{attribute 'linkalways'} 
{attribute 'no_explicit_call' := 'This FB is a CLASS and must be accessed using methods or properties'}
{attribute 'enable_dynamic_creation'}
FUNCTION_BLOCK FINAL Node_NOT EXTENDS Node
VAR
	in : _BOOL(FALSE);
	out : _BOOL(FALSE);
END_VAR

METHOD PUBLIC  Clone : I_Node
VAR
	pNode : POINTER TO Node_NOT;
END_VAR
pNode := __NEW(Node_NOT);
Clone := pNode^;
END_METHOD

METHOD FB_init : BOOL
VAR_INPUT
	bInitRetains : BOOL; // if TRUE, the retain variables are initialized (warm start / cold start)
	bInCopyCode : BOOL;  // if TRUE, the instance afterwards gets moved into the copy code (online change)
END_VAR
AddParameter('in', in);
AddOutput('out', out);

this^.Metadatum.AddBoolAsMetadata('deprecated', true);
END_METHOD

METHOD PROTECTED OnExecute
VAR
END_VAR
out.Value := NOT in.Value;
END_METHOD

END_FUNCTION_BLOCK

(* stored: Version 1.1.0.1, ProductVersion 3.1.4026.18
   POU Node_NOT: Id {d1c71ada-1c9a-09a5-235f-867c21a1fb89}, SpecialFunc None
   Folder Constructor: Id {d5bcdd98-fd22-0615-266b-837c2a4c7c32}
   Method Clone: Id {2fb93351-7500-0d11-041e-f8a77e39ea87}
   Method FB_init: Id {7336cfdf-b334-0c6a-384f-c02b9db6b810}
   Method OnExecute: Id {99c3b9b6-ab4e-08cd-3a91-7e75e73e5862} *)
